{attribute 'GeneratedUsingTerminal: EL9150--0000'}
{attribute addProperty BoxType "EL9150--0000"}
{attribute addProperty Description "EL9150 Power Supplier with LED(230V)"}
{attribute addProperty Physics "KK"}
{attribute addProperty Id "EL9150"}
{attribute addProperty CRC "2522918315"}
{attribute addProperty Size "0"}
TYPE EL9150_9660ADAB EXTENDS EtcSlaveTerminalBase_947E5A46 :
STRUCT
END_STRUCT
END_TYPE

(* stored: Version 1.2.0.0, ProductVersion 3.1.4024.9
   DUT EL9150_9660ADAB: Id {82a5dcd2-7c5d-49cb-ae33-f04d63e31332} *)
